{attribute 'linkalways'} 
{attribute 'no_explicit_call' := 'This FB is a CLASS and must be accessed using methods or properties'}
{attribute 'enable_dynamic_creation'}
FUNCTION_BLOCK ServerResponse IMPLEMENTS I_ServerResponse
VAR
	_header : Header(0);
	_sent : BOOL := FALSE;
	destination : REFERENCE TO ResponseData;
	config : I_ServerResponseConfig;
END_VAR

METHOD PUBLIC Accepted
VAR_INPUT
END_VAR
IF _sent THEN
	RETURN;
END_IF

config.UpdateResponseWithAccepted(THIS^);
SendHeaderToDestination();
END_METHOD

METHOD PUBLIC Busy
VAR_INPUT
END_VAR
IF _sent THEN
	RETURN;
END_IF

config.UpdateResponseWithBusy(THIS^);
SendHeaderToDestination();
END_METHOD

METHOD PUBLIC Error
VAR_INPUT
	Message : T_MAXSTRING;
END_VAR
IF _sent THEN
	RETURN;
END_IF

config.UpdateResponseWithError(THIS^, Message);
SendHeaderToDestination();
END_METHOD

METHOD FB_init : BOOL
VAR_INPUT
	bInitRetains : BOOL; // if TRUE, the retain variables are initialized (warm start / cold start)
	bInCopyCode : BOOL;  // if TRUE, the instance afterwards gets moved into the copy code (online change)
	Destination : REFERENCE TO ResponseData;
	Config : I_ServerResponseConfig;
END_VAR
THIS^.destination REF= Destination;
This^.config := Config;
END_METHOD

PROPERTY PUBLIC Header : I_Header
GET
Header := _header;
END_GET
END_PROPERTY

PROPERTY PUBLIC HeadersSent : BOOL
GET
HeadersSent := _sent;
END_GET
END_PROPERTY

METHOD PUBLIC Pending
VAR_INPUT
	ResponseId : T_MAXSTRING;
	RetryDelayInMs : UDINT;
END_VAR
IF _sent THEN
	RETURN;
END_IF

config.UpdateResponseWithPending(THIS^, ResponseId, RetryDelayInMs);
SendHeaderToDestination();
END_METHOD

METHOD PRIVATE SendHeaderToDestination
VAR_INPUT
END_VAR
_sent := TRUE;
_header.ToString(destination.Header);
END_METHOD

METHOD PUBLIC Success
VAR_INPUT
END_VAR
VAR
	errorMessage : T_MAXSTRING;
END_VAR
IF _sent THEN
	RETURN;
END_IF

config.UpdateResponseWithSuccess(THIS^);
SendHeaderToDestination();
memset(ADR(destination.Payload),0,SIZEOF(destination.Payload));
END_METHOD

METHOD PUBLIC SuccessWithPayload
VAR_INPUT
	PayloadDataAddress : PVOID;
	PayloadDataSize : UDINT;
END_VAR
VAR
	errorMessage : T_MAXSTRING;
END_VAR
IF _sent THEN
	RETURN;
END_IF

IF PayloadDataSize > SIZEOF(destination.Payload) THEN
	errorMessage := 'Payload too big to transmit. Maximum : ';
	errorMessage := concat(errorMessage, UDINT_TO_STRING(SIZEOF(destination.Payload)));
	errorMessage := concat(errorMessage, ', Actual Size : ');
	errorMessage := concat(errorMessage, UDINT_TO_STRING(SIZEOF(PayloadDataSize)));
	Error(errorMessage);
	RETURN;
END_IF

config.UpdateResponseWithSuccess(THIS^);
SendHeaderToDestination();
memcpy(ADR(destination.Payload),PayloadDataAddress,PayloadDataSize);
END_METHOD

END_FUNCTION_BLOCK

(* stored: Version 1.1.0.1, ProductVersion 3.1.4024.12
   POU ServerResponse: Id {01d8908d-0d42-4ebb-ab3f-dd0bcd0619c3}, SpecialFunc None
   Folder Constructor: Id {eecda43b-278b-4c0f-82ba-ef0138d22b11}
   Folder Private: Id {b6abcce5-8d92-4eee-bdc0-26f5665fa12d}
   Method Accepted: Id {6a11cffb-86d6-447b-9122-22fe8e08261c}
   Method Busy: Id {efb4c96f-8c99-484e-a56e-0f202efa6c3e}
   Method Error: Id {4133beb7-3ac7-45de-a9b6-b0641db40855}
   Method FB_init: Id {93971270-1190-4214-90ce-2458ab5b9410}
   Property Header: Id {1a5384de-2402-4919-b8b4-9eb07e9635aa}
   Get Get: Id {4d604038-9716-4bda-9a20-2c4af0caacb0}
   Property HeadersSent: Id {89071bf7-7d84-4f78-917f-6db1b9f33b9e}
   Get Get: Id {5e45cf4a-1c2f-444b-9783-839183a7d28a}
   Method Pending: Id {98b7607b-50e5-434a-a5ec-86c02f0b4693}
   Method SendHeaderToDestination: Id {c605e081-68c8-4516-bd6d-89fc22f16ff1}
   Method Success: Id {e8ec9304-2bdf-4fd2-9723-3f3b826dd538}
   Method SuccessWithPayload: Id {a0f936ba-3243-4794-876f-bbdda8e73d58} *)
